PROGRAM MAIN
VAR
	fbServo		: FB_Component_Servo;
	func		: INT;
	target		: INT := 50;
	set			: BOOL;
	hal			: BOOL;
	res			: BOOL;
	
	fbPiston	: FB_Component_DualValveGuarded;
	bEn: BOOL;
	
	tTimer		: TON;
END_VAR

fbPiston(sName := '',
	tTimeout := T#5S,
	bSensExtended := GVL.bWireClampTransverse2Extended,
	bSensRetracted := GVL.bWireClampTransverse2Retracted,
	bOutputA := GVL.bExtendWireHolderTransverse1,
	bOutputB := GVL.bRetractWireHolderTransverse1);

IF bEn AND NOT fbPiston.bEnabled THEN
	fbPiston.M_Enable();
	bEn := FALSE;
END_IF 

IF set THEN
	CASE func OF
		1: fbPiston.M_Extend();
		2: fbPiston.M_Retract();
		4: fbPiston.M_Halt();
		5: fbPiston.M_Resume();
		6: fbPiston.M_Disable();
	END_CASE
	set := FALSE;
END_IF



(*fbServo(
	sName 			:= '',
	tTimeout 		:= T#0MS,
	uMaxRPMservo 	:= 3000,
	rGearRatio 		:= 2.25,
	bRTO 			:= GVL.bReadyToOperate614,
	bEnableDrive 	:= GVL.b614Enable,
	bResetDrive 	:= GVL.bResetServosErrors,
	uAnalogOut 		:= GVL.aOutServo2);

IF NOT fbServo.bEnabled THEN
	fbServo.M_Enable();
END_IF

IF set THEN
	fbServo.M_SetAcceleration(uRPMperSec := 50);
	fbServo.M_SetRPMlimit(RPM := 700);
	fbServo.M_SetTargetRPM(target);
	set := FALSE;
END_IF

IF NOT GVL.bFeedBackSafetyRelay THEN
	IF NOT (fbServo.eState = E_State.HALTED) THEN
		fbServo.M_Halt();
		hal := FALSE;
	END_IF
	
END_IF

IF res THEN
	fbServo.M_Resume();
	res := FALSE;
END_IF*)

END_PROGRAM

(* stored: Version 1.1.0.1, ProductVersion 3.1.4024.15
   POU MAIN: Id {6907ca3e-912a-490f-aa07-3ae958d9385e}, SpecialFunc None *)
